{attribute 'linkalways'} 
{attribute 'no_explicit_call' := 'This FB is a CLASS and must be accessed using methods or properties'}
{attribute 'enable_dynamic_creation'}
FUNCTION_BLOCK FINAL XOR_ULINT EXTENDS Node
VAR
	in1 : _ULINT(0);
	in2 : _ULINT(0);
	out : _ULINT(0);
END_VAR

METHOD PUBLIC Clone : I_Node
VAR
	pNode : POINTER TO XOR_ULINT;
END_VAR
pNode := __NEW(XOR_ULINT);
Clone := pNode^;
END_METHOD

METHOD FB_init : BOOL
VAR_INPUT
	bInitRetains : BOOL; // if TRUE, the retain variables are initialized (warm start / cold start)
	bInCopyCode : BOOL;  // if TRUE, the instance afterwards gets moved into the copy code (online change)
END_VAR
AddInput('in1',THIS^.in1);
AddInput('in2',THIS^.in2);
AddOutput('out', THIS^.out);
END_METHOD

METHOD PROTECTED OnExecute
VAR
END_VAR
out.Value := in1.Value XOR in2.Value;
END_METHOD

END_FUNCTION_BLOCK

(* stored: Version 1.1.0.1, ProductVersion 3.1.4024.15
   POU XOR_ULINT: Id {68219f48-6d71-4541-802c-6ec232c20ac8}, SpecialFunc None
   Folder Constructor: Id {677fb147-15fd-4def-91b2-96dad0d5aada}
   Method Clone: Id {558d32dd-486f-4b4d-b916-29d98cd169d6}
   Method FB_init: Id {c4dd218e-0415-43b7-ab22-ea23ac2a278c}
   Method OnExecute: Id {66395bdc-8476-4f6f-8550-8bdc51247ef1} *)
